(* CoDeSys 2.3 export: DELAY.EXP *)

(* POU Components/Delay, ST *)
FUNCTION_BLOCK Delay
VAR_INPUT
	start:BOOL;
	stop:BOOL;
END_VAR
VAR_OUTPUT
END_VAR
VAR
	afterTime:BOOL;
	afterTimeImpulse:BOOL;
	untilTimePass:BOOL;
	counter: INT;
	timeSetup: INT;
END_VAR
IF NOT start  OR stop THEN
	counter := 0;
END_IF

IF clock1secImpulse AND start THEN
	counter := counter + 1;
END_IF
IF counter > timeSetup THEN
	counter := timeSetup;
END_IF

afterTimeImpulse:= NOT afterTime AND counter >= timeSetup;
afterTime := counter >= timeSetup;

untilTimePass := start AND (NOT stop) AND counter < timeSetup;
END_FUNCTION_BLOCK
